{attribute 'qualified_only'}
{attribute 'strict'}
TYPE e_TrackNum :
	(
	Big :=3,
	Small :=2,
	Main:=1	);	
END_TYPE

(* stored: Version 1.1.0.1, ProductVersion 3.1.4026.8
   DUT E_TrackNum: Id {8c7b446a-e63b-4ff3-8581-b59315de87a2} *)
